// Mitsubishi GX Works2 project: 0708-비교연산활용   PLC: Q02/Q02H

PROGRAM MAIN
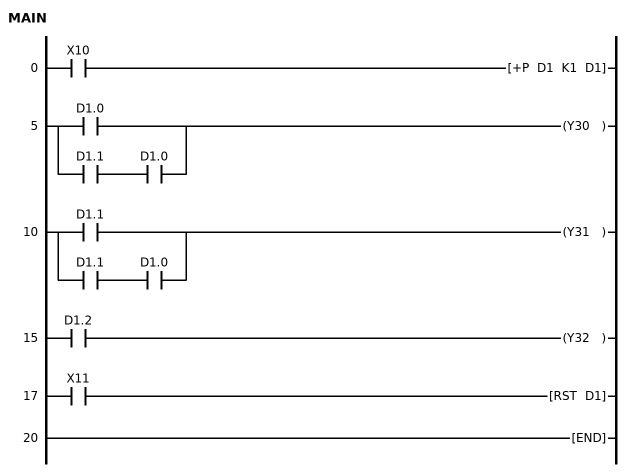
0     LD      X10
      +P      D1 K1 D1
5     LD      D1.0
      LD      D1.1
      AND     D1.0
      ORB
      OUT     Y30
10    LD      D1.1
      LD      D1.1
      AND     D1.0
      ORB
      OUT     Y31
15    LD      D1.2
      OUT     Y32
17    LD      X11
      RST     D1
20    END
END_PROGRAM
